# EPICS autosave request: ADApp/Db/pvCam_settings.req
$(P)$(R)GainX
$(P)$(R)GainY
$(P)$(R)Fidget
